FUNCTION_BLOCK FB_ConsumptionCalculator_Test EXTENDS TcUnit.FB_TestSuite
VAR_INPUT
END_VAR
VAR_OUTPUT
END_VAR
VAR
END_VAR

theCalculatedValueShouldBeTenAfterTenSeconds();
theCalculatedValueShouldBe20After20Seconds();
theCalulatedValueShouldBe30After20Seconds();

METHOD theCalculatedValueShouldBe20After20Seconds
VAR
	consumptionCalc : FB_ConsumptionCalculator;
END_VAR

TEST('theCalculatedValueShouldBe20After20Seconds');

consumptionCalc.calculate(
						start := TRUE,
						valuePerSec := 1,
						intervalMs := 10000,
						dtime := T#10S);
consumptionCalc.sum;								
consumptionCalc.calculate(
						start := TRUE,
						valuePerSec := 1,
						intervalMs := 10000,
						dtime := T#10S);
consumptionCalc.sum;			
						
AssertEquals_REAL(Expected := 20, Actual := consumptionCalc.sum, Delta := 0, Message := 'Calculated value not twenty after twenty seconds');

consumptionCalc.reset();
AssertEquals_REAL(Expected := 0, Actual := consumptionCalc.sum, Delta := 0, Message := 'Calculated value not reset');

TEST_FINISHED();
END_METHOD

METHOD theCalculatedValueShouldBeTenAfterTenSeconds : BOOL
VAR
	consumptionCalc : FB_ConsumptionCalculator;
END_VAR

TEST('theCalculatedValueShouldBeTenAfterTenSeconds');
consumptionCalc.calculate(
						start := TRUE,
						valuePerSec := 0,
						intervalMs := 10000,
						dtime := T#10MS);
	
consumptionCalc.sum;						
consumptionCalc.calculate(
						start := TRUE,
						valuePerSec := 1,
						intervalMs := 10000,
						dtime := T#10S);
consumptionCalc.sum;
						
AssertEquals_REAL(Expected := 10, Actual := consumptionCalc.sum, Delta := 0, Message := 'Calculated value not ten after ten seconds');

TEST_FINISHED();
END_METHOD

METHOD theCalulatedValueShouldBe30After20Seconds
VAR
	consumptionCalc : FB_ConsumptionCalculator;
END_VAR

TEST('theCalulatedValueShouldBe30After20Seconds');

consumptionCalc.calculate(
						start := TRUE,
						valuePerSec := 1,
						intervalMs := 10000,
						dtime := T#10S);
						
consumptionCalc.calculate(
						start := TRUE,
						valuePerSec := 2,
						intervalMs := 10000,
						dtime := T#10S);

AssertEquals_REAL(Expected := 30, Actual := consumptionCalc.sum, Delta := 0, Message := 'Calculated value not 30 after twenty seconds');


TEST_FINISHED();
END_METHOD

END_FUNCTION_BLOCK

(* stored: Version 1.1.0.1, ProductVersion 3.1.4024.9
   POU FB_ConsumptionCalculator_Test: Id {4e76fce4-8491-47f4-acc1-5379a12f6435}, SpecialFunc None
   Method theCalculatedValueShouldBe20After20Seconds: Id {4f57e544-87f9-4435-b2f8-17f180f6ac1a}
   Method theCalculatedValueShouldBeTenAfterTenSeconds: Id {2ce23a2a-5b79-4d69-b281-a57489cf4886}
   Method theCalulatedValueShouldBe30After20Seconds: Id {f24bc762-8013-4a64-adc3-55829c3371e4} *)
